KUKA KRL program: centerline_loop.src

&ACCESS RVP
&REL 1
&PARAM TEMPLATE = C:\KRC\Roboter\Template\vorgabe
DEF CENTERLINE_LOOP()

;PRESSURE GENERAL
CL_GunPressureCmd=405


;UPPER PIN RETRACT =  27252       RANGE 26000 - 28000
;UPPER PIN EXTENDED = 6602        RANGE 6500- 7000
;UPPER PIN WELD POSITION = 11674  RANGE 10000 - 13500


;GUN RETRACT = 139815             RANGE 137000 - 142000
;GUN EXTENDED = 61450             RANGE 60000 - 63000
;GUN WELD POSITION = 70915        RANGE 65000 - 76000


;FORMULA CMD = (MPa / 0.9) * 4095

;PRESSURE 455   0.10MPa    14.50 PSI
;PRESSURE 910   0.20MPa    29.01 PSI
;PRESSURE 1365  0.30MPa    43.51 PSI
;PRESSURE 1820  0.40MPa    58.02 PSI
;PRESSURE 2275  0.50MPa    72.52 PSI
;PRESSURE 2503  0.55MPa    79.77 PSI
;PRESSURE 2730  0.60MPa    87.02 PSI
LOOP

$OUT[472]=FALSE
$OUT[471]=TRUE
$OUT[498]=FALSE
$OUT[499]=TRUE
$OUT[501]=FALSE
$OUT[502]=TRUE
$OUT[495]=FALSE
$OUT[496]=TRUE
$OUT[503]=FALSE
$OUT[504]=TRUE
$OUT[494]=FALSE
$OUT[500]=FALSE
$OUT[505]=FALSE
$OUT[473]=FALSE

WAIT FOR $IN[482]
WAIT SEC 1.0

$OUT[504]=FALSE
WAIT SEC 0.2
$OUT[503]=TRUE
WAIT FOR $IN[470]
WAIT SEC 0.5

$OUT[496]=FALSE
WAIT SEC 0.2
$OUT[495]=TRUE
WAIT SEC 0.50

$OUT[503]=FALSE
WAIT SEC 0.2
$OUT[504]=TRUE
WAIT FOR $IN[482]
WAIT SEC 0.5

$OUT[499]=FALSE
WAIT SEC 0.2
$OUT[498]=TRUE
WAIT SEC 0.5

$OUT[502]=FALSE
WAIT SEC 0.2
$OUT[501]=TRUE
WAIT SEC 0.5

$OUT[471]=FALSE
WAIT SEC 0.2
$OUT[472]=TRUE
WAIT SEC 1.0

$OUT[495]=FALSE
WAIT SEC 0.2
$OUT[496]=TRUE
WAIT SEC 0.5

$OUT[472]=FALSE
WAIT SEC 0.2
$OUT[471]=TRUE
WAIT SEC 1.0

$OUT[501]=FALSE
WAIT SEC 0.2
$OUT[502]=TRUE
WAIT SEC 0.5

$OUT[498]=FALSE
WAIT SEC 0.2
$OUT[499]=TRUE
WAIT SEC 1.0

$OUT[504]=TRUE
$OUT[496]=TRUE

WAIT FOR $IN[482]
WAIT SEC 2.0

ENDLOOP
END
